(* CoDeSys 2.3 export: 1.EXP *)
(* Libraries: Standard.lib 2.12.10 15:48:34, SYSLIBCALLBACK.LIB 2.12.10 15:48:32 *)

(* PLC configuration (modules and I/O channels)
Hardware configuration [Root] node -1, in %IB0 out %QB0
  K-Bus [K_Bus] node 0, in %IB0 out %QB0
    0750-1504 16 DO 24V DC 0.5A [Type_10_16_Channels] node 0, in %IB0 out %QB0 {param 10000 = PLC; param 10001 = plugged}
      AT %QX0.0 [BOOLOnX_Q] Ch_1 Digital output
      AT %QX0.1 [BOOLOnX_Q] Ch_2 Digital output
      AT %QX0.2 [BOOLOnX_Q] Ch_3 Digital output
      AT %QX0.3 [BOOLOnX_Q] Ch_4 Digital output
      AT %QX0.4 [BOOLOnX_Q] Ch_5 Digital output
      AT %QX0.5 [BOOLOnX_Q] Ch_6 Digital output
      AT %QX0.6 [BOOLOnX_Q] Ch_7 Digital output
      AT %QX0.7 [BOOLOnX_Q] Ch_8 Digital output
      AT %QX0.8 [BOOLOnX_Q] Ch_9 Digital output
      AT %QX0.9 [BOOLOnX_Q] Ch_10 Digital output
      AT %QX0.10 [BOOLOnX_Q] Ch_11 Digital output
      AT %QX0.11 [BOOLOnX_Q] Ch_12 Digital output
      AT %QX0.12 [BOOLOnX_Q] Ch_13 Digital output
      AT %QX0.13 [BOOLOnX_Q] Ch_14 Digital output
      AT %QX0.14 [BOOLOnX_Q] Ch_15 Digital output
      AT %QX0.15 [BOOLOnX_Q] Ch_16 Digital output
  Fieldbus variables [FB_VARS] node 1, in %IB0 out %QB0
  Flag variables [FLAG_VARS] node 2, in %IB0 out %QB0
  Modbus-Master [MB_MASTER] node 3, in %IB0 out %QB0
*)

(* POU PLC_PRG, ST *)
PROGRAM PLC_PRG
VAR
	var1: INT;
END_VAR
var1:= 10;
END_PROGRAM
